PROGRAM main
VAR
	Remote_Start AT %IX0.2 : bool;
	Local_Start AT %IX0.3 : bool;
	Motor_1 AT %QX0.1 : bool;
END_VAR

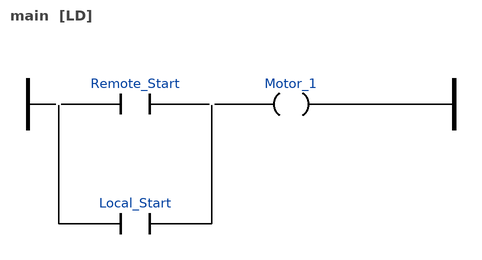
(* LD diagram, written out as Structured Text *)
Motor_1 := Remote_Start OR Local_Start;
END_PROGRAM
